FUNCTION_BLOCK PUBLIC PAEMisalignment EXTENDS PAESensorDigital
VAR_INPUT
END_VAR
VAR_OUTPUT
END_VAR
VAR
END_VAR

END_FUNCTION_BLOCK

(* stored: Version 1.1.0.1, ProductVersion 3.1.4020.6
   POU PAEMisalignment: Id {2d09b40c-cd02-401a-84da-779eeb4b2dbe}, SpecialFunc None *)
